SYSTEM IcaruDelay (* System Configuration *)
  (* Standard: 61499-1 *)
  (* Version 0.4, 2009-03-05, JHC, Holobloc Inc., Deleted Application. *)
  (* Version 0.3, 2003-12-05, JHC, Rockwell Automation, Renamed from NEWSYSTEM. *)
  (* Version 0.2, 2002-11-05, JHC, Rockwell Automation, Fixed missing (empty) FBD in Application. *)
  (* Version 0.1, 2002-01-17, JHC, Rockwell Automation, Minor cleanup *)
  (* Version 0.0, 2000-05-27, JHC, Rockwell Automation *)
  DEVICE ICARU4442 : RMT_DEV(MGR_ID := "localhost:61494")
    RESOURCE RESM : EMB_RES
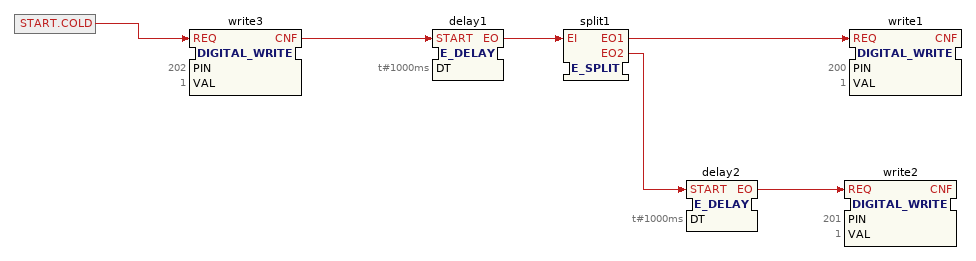
      FBS
        write1 : DIGITAL_WRITE(PIN := 200, VAL := 1);
        write2 : DIGITAL_WRITE(PIN := 201, VAL := 1);
        delay1 : E_DELAY(DT := t#1000ms);
        delay2 : E_DELAY(DT := t#1000ms);
        split1 : E_SPLIT;
        write3 : DIGITAL_WRITE(PIN := 202, VAL := 1);
      END_FBS
      EVENT_CONNECTIONS
        delay1.EO TO split1.EI;
        split1.EO1 TO write1.REQ;
        split1.EO2 TO delay2.START;
        delay2.EO TO write2.REQ;
        START.COLD TO write3.REQ;
        write3.CNF TO delay1.START;
      END_CONNECTIONS
    END_RESOURCE
  END_DEVICE
END_SYSTEM
